ABB RobotStudio station: Est_5.rsstn

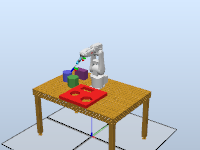
Station Solution_1_Tutorial (saved by RobotStudio 20.1.9056.2)
Controller Controller1, task T_ROB1: task frame (RAPID world) sits at (0, 150, 830) mm, rotated rx 0 ry 0 rz -90 deg in the station
Controller Controller1
  mechanical unit ROB_1: IRB120_3_58__01, 6 joints, base frame (0, 0, 0) mm
Layout (positions relative to the parent item):
  - table [part] at (-200, -500, 830) mm
  - object_1 [part] at (-600, -150, 830) mm
  - object_2 [part] at (-650, -150, 830) mm
  - object_3 [part] at (-700, -200, 830) mm
  - siegmund_1500_1000 [part]
  - object_11 [part] at (-200, -500, 830) mm
  - object_22 [part] at (-200, -500, 830) mm
  - object_33 [part] at (-200, -500, 830) mm
  - smc_gripper [mechanism, from Libraries\smc_gripper.rslib] at (0, -214.35, 1424) mm, rotated rx 180 ry 60 rz 90 deg
  - IRB120_3_58__01 [mechanism, from Robots\IRB120_3_58_G_01.rslib] at (0, 150, 830) mm, rotated rx 0 ry 0 rz -90 deg; joint values [0, 0, 0, 0, 0.5236, 0] (rad or m)
  - Positioner_obj_1 [smart component, from Components\Positioner.rslib]
      properties: Object=object_1; Position=[-0.6 -0.15 0.83]; Orientation=[0 0 0]; Reference=Global; ReferenceObject=(none)
  - Positioner_obj_2 [smart component, from Components\Positioner.rslib]
      properties: Object=object_2; Position=[-0.65 -0.15 0.83]; Orientation=[0 0 0]; Reference=Global; ReferenceObject=(none)
  - Positioner_obj_3 [smart component, from Components\Positioner.rslib]
      properties: Object=object_3; Position=[-0.7 -0.2 0.83]; Orientation=[0 0 0]; Reference=Global; ReferenceObject=(none)
  - Attacher_obj_1 [smart component, from Components\Attacher.rslib]
      properties: Parent=smc_gripper; Flange=0; Child=object_1; Mount=false; Offset=[0 0 0]; Orientation=[0 0 0]
  - Attacher_obj_2 [smart component, from Components\Attacher.rslib]
      properties: Parent=smc_gripper; Flange=0; Child=object_2; Mount=false; Offset=[0 0 0]; Orientation=[0 0 0]
  - Attacher_obj_3 [smart component, from Components\Attacher.rslib]
      properties: Parent=smc_gripper; Flange=0; Child=object_3; Mount=false; Offset=[0 0 0]; Orientation=[0 0 0]
  - Detacher_obj_1 [smart component, from Components\Detacher.rslib]
      properties: Child=object_1; KeepPosition=true
  - Detacher_obj_3 [smart component, from Components\Detacher.rslib]
      properties: Child=object_3; KeepPosition=true
  - Detacher_obj_2 [smart component, from Components\Detacher.rslib]
      properties: Child=object_2; KeepPosition=true
Attachment: smc_gripper is attached to IRB120_3_58__01 / Link6
Station signals: DI object_1_positioner, DI object_2_positioner, DI object_3_positioner
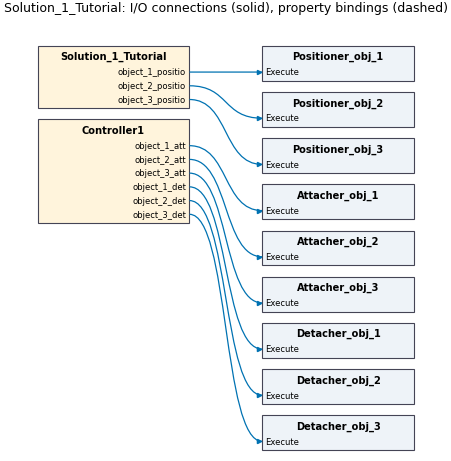
Station logic (signal -> signal, property => property):
  Solution_1_Tutorial.object_1_positioner -> Positioner_obj_1.Execute
  Solution_1_Tutorial.object_2_positioner -> Positioner_obj_2.Execute
  Solution_1_Tutorial.object_3_positioner -> Positioner_obj_3.Execute
  Controller1.object_1_att -> Attacher_obj_1.Execute
  Controller1.object_2_att -> Attacher_obj_2.Execute
  Controller1.object_3_att -> Attacher_obj_3.Execute
  Controller1.object_1_det -> Detacher_obj_1.Execute
  Controller1.object_2_det -> Detacher_obj_2.Execute
  Controller1.object_3_det -> Detacher_obj_3.Execute
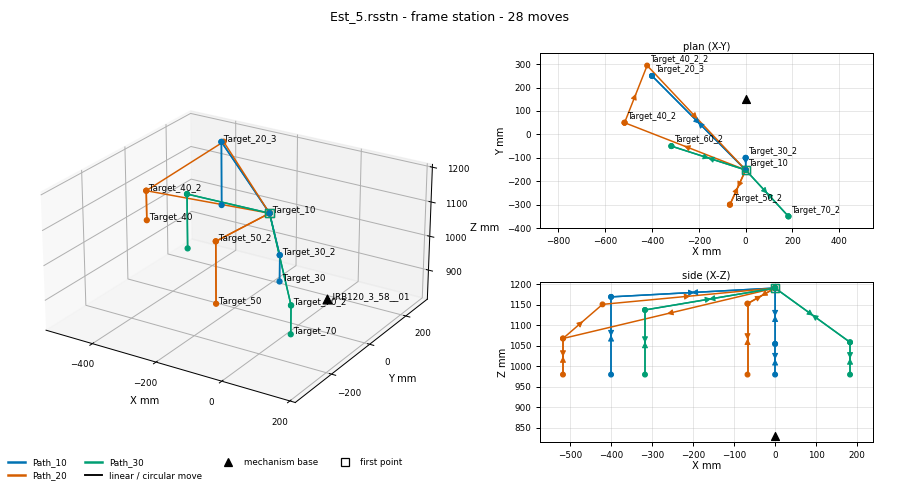
[picture p0: tool path of Est_5.rsstn in frame station, 28 of 28 moves have a stored position in this frame; points joined in program order, loops and branches not executed]
Targets, tools, work objects and paths stored in the station, written as RAPID:
! task T_ROB1
MODULE CalibData
  PERS tooldata smc_gripper:=[TRUE,[[0,0.004,197.001],[1,0,0,0]],[1,[0.207,-0.496,71.18],[1,0,0,0],0,0,0]];
ENDMODULE

! task T_ROB1
MODULE Module1
  CONST robtarget Target_10:=[[302,0.004,360.999],[0,0,1,0],[-1,0,-1,0],[9E+09,9E+09,9E+09,9E+09,9E+09,9E+09]];
  CONST robtarget Target_20:=[[-100,-400,150],[0,0,1,0],[-2,0,-2,0],[9E+09,9E+09,9E+09,9E+09,9E+09,9E+09]];
  CONST robtarget Target_20_3:=[[-100,-400,339.482109829],[0,0,1,0],[-2,0,-2,0],[9E+09,9E+09,9E+09,9E+09,9E+09,9E+09]];
  CONST robtarget Target_30:=[[250,0,150],[0,0,1,0],[-1,0,-1,0],[9E+09,9E+09,9E+09,9E+09,9E+09,9E+09]];
  CONST robtarget Target_30_2:=[[250,0,224.88153549],[0,0,1,0],[-1,0,-1,0],[9E+09,9E+09,9E+09,9E+09,9E+09,9E+09]];
  CONST robtarget Target_40:=[[100,-517.298,150],[0,0,1,0],[-1,0,-1,0],[9E+09,9E+09,9E+09,9E+09,9E+09,9E+09]];
  CONST robtarget Target_40_2:=[[100,-517.298,237.997639317],[0,0,1,0],[-1,0,-1,0],[9E+09,9E+09,9E+09,9E+09,9E+09,9E+09]];
  CONST robtarget Target_50:=[[450,-67.298,150],[0,0,1,0],[-1,0,-1,0],[9E+09,9E+09,9E+09,9E+09,9E+09,9E+09]];
  CONST robtarget Target_50_2:=[[450,-67.298,322.949199197],[0,0,1,0],[-1,0,-1,0],[9E+09,9E+09,9E+09,9E+09,9E+09,9E+09]];
  CONST robtarget Target_60:=[[200,-317.298,150],[0,0,1,0],[-1,0,-1,0],[9E+09,9E+09,9E+09,9E+09,9E+09,9E+09]];
  CONST robtarget Target_60_2:=[[200,-317.298,307.543483677],[0,0,1,0],[-1,0,-1,0],[9E+09,9E+09,9E+09,9E+09,9E+09,9E+09]];
  CONST robtarget Target_70:=[[500,182.702,150],[0,0,1,0],[0,0,0,0],[9E+09,9E+09,9E+09,9E+09,9E+09,9E+09]];
  CONST robtarget Target_70_2:=[[500,182.702,228.799643124],[0,0,1,0],[0,0,0,0],[9E+09,9E+09,9E+09,9E+09,9E+09,9E+09]];
  CONST robtarget Target_40_2_2:=[[-144.23137906,-420.892869102,321.185791052],[0,0,1,0],[-2,0,-2,0],[9E+09,9E+09,9E+09,9E+09,9E+09,9E+09]];
  PROC Path_10()
    MoveL Target_10,v100,z100,smc_gripper\WObj:=wobj0;
    MoveL Target_20_3,v100,z100,smc_gripper\WObj:=wobj0;
    MoveL Target_20,v100,fine,smc_gripper\WObj:=wobj0;
    PulseDO object_1_att;
    WaitTime 1;
    MoveL Target_20_3,v100,fine,smc_gripper\WObj:=wobj0;
    MoveL Target_10,v100,z100,smc_gripper\WObj:=wobj0;
    MoveL Target_30_2,v100,z100,smc_gripper\WObj:=wobj0;
    MoveL Target_30,v100,fine,smc_gripper\WObj:=wobj0;
    PulseDO object_1_det;
    WaitTime 1;
    MoveL Target_30_2,v100,fine,smc_gripper\WObj:=wobj0;
    MoveL Target_10,v100,z100,smc_gripper\WObj:=wobj0;
  ENDPROC
  PROC Path_20()
    MoveL Target_10,v100,z100,smc_gripper\WObj:=wobj0;
    MoveL Target_40_2,v100,z100,smc_gripper\WObj:=wobj0;
    MoveL Target_40,v100,fine,smc_gripper\WObj:=wobj0;
    PulseDO object_2_att;
    WaitTime 1;
    MoveL Target_40_2,v100,fine,smc_gripper\WObj:=wobj0;
    MoveL Target_40_2_2,v100,z100,smc_gripper\WObj:=wobj0;
    MoveL Target_10,v100,z100,smc_gripper\WObj:=wobj0;
    MoveL Target_50_2,v100,z100,smc_gripper\WObj:=wobj0;
    MoveL Target_50,v100,fine,smc_gripper\WObj:=wobj0;
    PulseDO object_2_det;
    WaitTime 1;
    MoveL Target_50_2,v100,fine,smc_gripper\WObj:=wobj0;
    MoveL Target_10,v100,z100,smc_gripper\WObj:=wobj0;
  ENDPROC
  PROC Path_30()
    MoveL Target_10,v100,z100,smc_gripper\WObj:=wobj0;
    MoveL Target_60_2,v100,z100,smc_gripper\WObj:=wobj0;
    MoveL Target_60,v100,fine,smc_gripper\WObj:=wobj0;
    PulseDO object_3_att;
    WaitTime 1;
    MoveL Target_60_2,v100,fine,smc_gripper\WObj:=wobj0;
    MoveL Target_10,v100,z100,smc_gripper\WObj:=wobj0;
    MoveL Target_70_2,v100,z100,smc_gripper\WObj:=wobj0;
    MoveL Target_70,v100,fine,smc_gripper\WObj:=wobj0;
    PulseDO object_3_det;
    WaitTime 1;
    MoveL Target_70_2,v100,fine,smc_gripper\WObj:=wobj0;
    MoveL Target_10,v100,z100,smc_gripper\WObj:=wobj0;
  ENDPROC
ENDMODULE

